{attribute 'GeneratedUsingTerminal: EL9560-0000-0016'}
{attribute addProperty BoxType "EL9560-0000-0016"}
{attribute addProperty Id "Status_UsAT %I*Status_Us_449D6AB51Status_UoAT %I*Status_Uo_449D6AB51WcStateAT %I*WcState_9091E0EB2InfoDataAT %I*InfoData_6F19DB2B2"}
{attribute addProperty CRC "3712328458"}
{attribute addProperty Size "6"}
TYPE EL9560_DD45A30A EXTENDS EtcSlaveTerminalBase_947E5A46 :
STRUCT
	{attribute addProperty Name "Status_Us"}
	Status_Us : Status_Us_449D6AB5;
	{attribute addProperty Name "Status_Uo"}
	Status_Uo : Status_Uo_449D6AB5;
	{attribute addProperty Name "WcState"}
	WcState : WcState_9091E0EB;
	{attribute addProperty Name "InfoData"}
	InfoData : InfoData_6F19DB2B;
END_STRUCT
END_TYPE

(* stored: Version 1.2.0.0, ProductVersion 3.1.4024.9
   DUT EL9560_DD45A30A: Id {910c9262-4594-46ba-b2ac-eb5fc6032c13} *)
